# EPICS autosave request: ADApp/Db/NDPluginBase_settings.req
$(P)$(R)NDArrayPort
$(P)$(R)NDArrayAddress
$(P)$(R)EnableCallbacks
$(P)$(R)MinCallbackTime
$(P)$(R)BlockingCallbacks
$(P)$(R)QueueSize
$(P)$(R)NumThreads
file "NDArrayBase_settings.req", P=$(P), R=$(R)
